// Core §8.10: shelving suppresses ANNUNCIATION only. Unrationalized -> refuse;
// SAFETY -> refuse; a shelved MANUAL_RESET alarm STILL BLOCKS (the O7 test).
// Auto-expiry timing is runtime-verified (F_Now-driven).
FUNCTION_BLOCK FB_Shelve_Tests EXTENDS TcUnit.FB_TestSuite
VAR
    _log : FB_AlarmLog;
    _s1, _s2, _s3, _s4 : INT;
    _w : BOOL;
END_VAR

IF NOT _w THEN
    _log.RegisterMeta(Reason := 100, OperatorAction := 'act', Consequence := 'cons', Shelvable := TRUE);
    _s1 := _log.Raise(Reason := 100, Text := 'shelvable blocking',
        Source := 'T', Severity := E_Severity.HIGH, Category := E_Category.PROCESS,
        ResetClass := E_ResetClass.MANUAL_RESET);
    _s2 := _log.Raise(Reason := 200, Text := 'no meta',
        Source := 'T', Severity := E_Severity.LOW, Category := E_Category.PROCESS,
        ResetClass := E_ResetClass.AUTO_RESET);
    _s3 := _log.Raise(Reason := 300, Text := 'safety',
        Source := 'T', Severity := E_Severity.HIGH, Category := E_Category.SAFETY,
        ResetClass := E_ResetClass.MANUAL_RESET);
    _s4 := _log.Raise(Reason := E_Reason.TASK_JITTER_HIGH, Text := 'generated',
        Source := 'T', Severity := E_Severity.HIGH, Category := E_Category.PROCESS,
        ResetClass := E_ResetClass.AUTO_RESET);
    _w := TRUE;
END_IF
Unrationalized_refused();
Safety_refused();
Zero_duration_refused();
Shelved_still_blocks();
Generated_metadata_is_authoritative();
Reused_slot_clears_shelf_state();

METHOD Unrationalized_refused
TEST('Unrationalized_refused');
AssertFalse(Condition := _log.Shelve(Slot := _s2, DurationS := 60),
            Message := 'no rationalization record -> not shelvable (§8.10)');
TEST_FINISHED();
END_METHOD

METHOD Generated_metadata_is_authoritative
TEST('Generated_metadata_is_authoritative');
AssertEquals_DINT(Expected := TO_DINT(E_Severity.LOW),
    Actual := TO_DINT(_log.Active[_s4].Severity),
    Message := 'generated priority replaces caller reclassification');
AssertEquals_DINT(Expected := TO_DINT(E_Category.SYSTEM),
    Actual := TO_DINT(_log.Active[_s4].Category),
    Message := 'generated class replaces caller reclassification');
AssertTrue(Condition := _log.Shelve(Slot := _s4, DurationS := 60),
    Message := 'generated shelvability needs no project registration');
AssertFalse(Condition := _log.RegisterMeta(Reason := E_Reason.TASK_JITTER_HIGH,
    OperatorAction := 'override', Consequence := 'override', Shelvable := FALSE),
    Message := 'standard metadata cannot be overridden per project');
AssertFalse(Condition := _log.RegisterMetaFull(Reason := 400,
    OperatorAction := 'act', Consequence := '', Priority := E_Severity.LOW,
    Category := E_Category.PROCESS, Shelvable := FALSE),
    Message := 'external metadata requires a complete consequence');
AssertFalse(Condition := _log.RegisterMetaFull(Reason := 401,
    OperatorAction := 'act', Consequence := 'cons', Priority := 99,
    Category := E_Category.PROCESS, Shelvable := FALSE),
    Message := 'external priority ordinal is bounds checked');
AssertFalse(Condition := _log.RegisterMetaFull(Reason := 402,
    OperatorAction := 'act', Consequence := 'cons', Priority := E_Severity.HIGH,
    Category := E_Category.SAFETY, Shelvable := TRUE),
    Message := 'external Safety metadata cannot enable shelving');
_log.Unshelve(Slot := _s4);
_log.Gone(Slot := _s4);
TEST_FINISHED();
END_METHOD

METHOD Zero_duration_refused
TEST('Zero_duration_refused');
AssertFalse(Condition := _log.Shelve(Slot := _s1, DurationS := 0),
            Message := 'zero-duration shelf cannot become permanent (8.10)');
TEST_FINISHED();
END_METHOD

METHOD Safety_refused
TEST('Safety_refused');
_log.RegisterMeta(Reason := 300, OperatorAction := 'x', Consequence := 'y', Shelvable := TRUE);
AssertFalse(Condition := _log.Shelve(Slot := _s3, DurationS := 60),
            Message := 'SAFETY category never shelvable, even flagged (§8.10)');
TEST_FINISHED();
END_METHOD

METHOD Reused_slot_clears_shelf_state
VAR
    slot : INT;
END_VAR
TEST('Reused_slot_clears_shelf_state');
AssertTrue(Condition := _log.Shelve(Slot := _s1, DurationS := 60), Message := 'shelf before close');
_log.Gone(Slot := _s1);
_log.OperatorReset();
slot := _log.Raise(Reason := 100, Text := 'reused slot',
    Source := 'T', Severity := E_Severity.LOW, Category := E_Category.PROCESS,
    ResetClass := E_ResetClass.AUTO_RESET);
AssertFalse(Condition := _log.Active[slot].Shelved,
            Message := 'new event never inherits a prior occupant shelf');
_log.Gone(Slot := slot);
TEST_FINISHED();
END_METHOD

METHOD Shelved_still_blocks
TEST('Shelved_still_blocks');
AssertTrue(Condition := _log.Blocking, Message := 'MANUAL_RESET alarm blocks before shelve');
AssertTrue(Condition := _log.Shelve(Slot := _s1, DurationS := 60), Message := 'rationalized+flagged shelves OK');
AssertTrue(Condition := _log.Active[_s1].Shelved, Message := 'annunciation suppressed');
AssertTrue(Condition := _log.Blocking, Message := 'STILL BLOCKING while shelved - control untouched (O7)');
AssertTrue(Condition := _log.Unshelve(Slot := _s1), Message := 'unshelve restores');
AssertFalse(Condition := _log.Active[_s1].Shelved, Message := 'flag cleared');
TEST_FINISHED();
END_METHOD

END_FUNCTION_BLOCK

(* stored: Version 1.1.0.1, ProductVersion 3.1.4024.12
   POU FB_Shelve_Tests: Id {721646f8-235c-463c-87d0-81c13f121fd7}, SpecialFunc None
   Method Unrationalized_refused: Id {1af6cabb-12b7-494d-bfe3-7029612c6294}
   Method Generated_metadata_is_authoritative: Id {b6840889-622d-4989-b43b-5c25ea446768}
   Method Zero_duration_refused: Id {6b354a8a-a05f-4488-b38e-f37b2c35d487}
   Method Safety_refused: Id {61359fa1-77ff-4c8e-a2d0-62816e5e6055}
   Method Reused_slot_clears_shelf_state: Id {33df6889-a2b4-421c-acd2-204122c864d1}
   Method Shelved_still_blocks: Id {3de61e9c-2bcd-483f-ba89-06703432aee1} *)
